(* CODESYS project sysprocess.20211125.1.project

Project tree, tasks and I/O mapping:
  MIC7001 : Changsha-Cyber-MI-linux, Changsha Cyber-MI Co., Ltd., version 3.5.10.40
    application Application
      libraries: Standard, * (System); CAA Types Extern, * (CAA Technical Workgroup); CAA Callback Extern, * (CAA Technical Workgroup); SysMem, * (System); SysTypes Interfaces, * (System); SysTime, * (System); CAA DTUtil Extern, 3.5.12.0 (CAA Technical Workgroup); CAA Real Time Clock Extern, 3.5.10.0 (CAA Technical Workgroup); CAN API, 1.0.0.3 (3S - Smart Software Solutions GmbH); SysFile, 3.5.15.0 (System); AC_DataLog, 3.5.14.0 (3S - Smart Software Solutions GmbH); CAA Net Base Services, 3.5.15.0 (CAA Technical Workgroup); CAA Memory, 3.5.12.0 (CAA Technical Workgroup); CAA SerialCom, 3.5.15.0 (CAA Technical Workgroup); Util, 3.5.15.0 (System); CAA Can Low Level Imp Extern, 3.5.11.0 (CAA Technical Workgroup); CAA Can Low Level Extern, 3.5.15.0 (CAA Technical Workgroup); VisuDialogs, * (System); CmpBitmapPool, * (System); CAA File, 3.5.15.0 (CAA Technical Workgroup); IODrvEtherCAT, 3.5.15.50 (3S - Smart Software Solutions GmbH); SysShm Implementation, 3.5.16.0 (System); SysShm, 3.5.8.0 (System); MIC7001 base library, 1.11 (Cyber-MI.com); CmpPlcShell, 3.5.5.0 (3S - Smart Software Solutions GmbH); SysProcess, 3.5.7.0 (System); CmpErrors2 Interfaces, 3.5.15.0 (System)
      task Task_20ms (cyclic, interval t#20ms, priority 10) calls prg_syscommand
      program prg_syscommand [ST]
    SoftMotion General Axis Pool
  libraries: CmpBitmapPool, * (System)
  5ce3da45-db07-42e7-a21c-a00fff4ed8f6|D:\工作文件\009中集集团\DOCS\等油耗图.jpg
  5ce3da45-db07-42e7-a21c-a00fff4ed8f6|C:\Users\RJST\Desktop\bmp1.png
  text list GlobalTextList
*)

// MIC7001/Application/prg_syscommand
PROGRAM prg_syscommand
VAR  
	syscmd:STRING(255);
	rst : RTS_IEC_RESULT;
	free_m:STRING(255);
	disk_userapp:DINT;
	disk_userdata:DINT;
	xGetFreeDisk :BOOL := FALSE;
END_VAR


// need to add the 2 line below into codesys config file(CODESYSConfig.cfg)

// [SysProcess]
// Command=AllowAll

IF xGetFreeDisk THEN
	syscmd := 'df -m|grep userapp |awk $'{print $$4} $'';
	sysprocess.SysProcessExecuteCommand2(pszCommand := syscmd, pszStdOut := free_m, udiStdOutLen := 255, pResult := ADR(rst) );
	disk_userapp := ANY_TO_DINT(free_m);
	
	syscmd := 'df -m|grep userdata |awk $'{print $$4} $'';
	sysprocess.SysProcessExecuteCommand2(pszCommand := syscmd, pszStdOut := free_m, udiStdOutLen := 255, pResult := ADR(rst) );
	disk_userdata := ANY_TO_DINT(free_m);
	xGetFreeDisk := FALSE;
END_IF

END_PROGRAM
